TYPE SSI_Encoder :
STRUCT
	uCounterValue	: UDINT ;		// Raw counter value
	rScaled			: REAL ;		// scaled value
	bDataError		: BOOL ;		
	bFrameError		: BOOL ;
	bPowerFailure	: BOOL ;
	bDataMismatch	: BOOL ;
	bSyncError		: BOOL ;
	bPDO_State		: BOOL ;
	bPDO_Toggle		: BOOL ;
END_STRUCT
END_TYPE

(* stored: Version 1.1.0.1, ProductVersion 3.1.4024.12
   DUT SSI_Encoder: Id {72802ae4-d0ca-4a3e-a1bf-6a7ca1ea7535} *)
